// TIA Portal V17 export
// export: Created 2025-03-10T13:12:12.59676Z, ExportSetting WithDefaults, DisplayName Totally Integrated Automation Portal, DisplayVersion V17 Update 8, DisplayName TIA Portal Openness, DisplayVersion V17 Update 8, DisplayName TIA Portal Version Control Interface, DisplayVersion V17, DisplayName SINAMICS Startdrive Advanced, DisplayVersion V17 SP2, DisplayName SINAMICS Startdrive G110M, G120, G120C, G120D, G120P, G115D, DisplayVersion V17 SP2, DisplayName SINAMICS Startdrive G130, G150, S120, S150, SINAMICS MV, S210, DisplayVersion V17 SP2, DisplayName STEP 7 Professional, DisplayVersion V17 Update 8, DisplayName SINUMERIK ONE STEP 7 Toolbox, DisplayVersion V17 Update 12, DisplayName SINUMERIK 840D sl STEP 7 Toolbox, DisplayVersion V17 Update 12, DisplayName STEP 7 Safety, DisplayVersion V17 Update 6, DisplayName WinCC Advanced, DisplayVersion V17 Update 8
TYPE "LIOLink_typeDiagnostics"
// stored: IsFailsafeCompliant false
   STRUCT
      status { ExternalVisible := 'False'; ExternalWritable := 'False'} : Word;   // Status of the Block or error identification when error occurred
      subfunctionStatus { ExternalVisible := 'False'; ExternalWritable := 'False'} : DWord;   // Status or return value of called FB's, FCs and system blocks
      stateNumber { ExternalVisible := 'False'; ExternalWritable := 'False'} : DInt;   // State in the state machine of the block where the error occurred
   END_STRUCT;
END_TYPE
